INTERFACE I_EventArguments EXTENDS I_Base

METHOD AddString : I_EventArguments
VAR_INPUT
	Argument : STRING;
END_VAR
END_METHOD

METHOD Clear : I_EventArguments
VAR_INPUT
END_VAR
END_METHOD

END_INTERFACE

(* stored: Version 1.1.0.1, ProductVersion 3.1.4026.18
   Itf I_EventArguments: Id {5fe54d5b-6bc7-4222-856f-4263dbc1a30a}
   Method AddString: Id {54bf0031-ba16-4d7e-be75-fc922e00da46}
   Method Clear: Id {9dd9def1-3051-4b42-a743-6d6d2fdf370b} *)
